{attribute 'OPC.UA.DA.StructuredType' := '1'}
{attribute 'OPC.UA.DA' := '1'}
TYPE stVisStatusAMR :
STRUCT
	State:  eState;
	Mode: eMode;
	isMoving: BOOL;
	isReady: BOOL;
	isConnected: BOOL;
// 	isLocked: BOOL;
	isBusy: BOOL;
	
	isDocked: BOOL;
	TargetReached: BOOL;
	isInCollision: BOOL;
	hasError: BOOL;
	TCPPosition: stPose2D;
END_STRUCT
END_TYPE

(* stored: Version 1.1.0.1, ProductVersion 3.1.4026.18
   DUT stVisStatusAMR: Id {bc669fa9-d258-45ab-8cb5-80efaf1ca196} *)
